// TIA Portal V17 export
// export: Created 2025-03-05T07:59:25.5463254Z, ExportSetting WithDefaults, DisplayName Totally Integrated Automation Portal, DisplayVersion V17 Update 8, DisplayName TIA Portal Openness, DisplayVersion V17 Update 8, DisplayName TIA Portal Version Control Interface, DisplayVersion V17, DisplayName SINAMICS Startdrive Advanced, DisplayVersion V17 SP2, DisplayName SINAMICS Startdrive G110M, G120, G120C, G120D, G120P, G115D, DisplayVersion V17 SP2, DisplayName SINAMICS Startdrive G130, G150, S120, S150, SINAMICS MV, S210, DisplayVersion V17 SP2, DisplayName STEP 7 Professional, DisplayVersion V17 Update 8, DisplayName SINUMERIK ONE STEP 7 Toolbox, DisplayVersion V17 Update 12, DisplayName SINUMERIK 840D sl STEP 7 Toolbox, DisplayVersion V17 Update 12, DisplayName STEP 7 Safety, DisplayVersion V17 Update 6, DisplayName WinCC Advanced, DisplayVersion V17 Update 8
FUNCTION "FC8001_PART_CHANGE" : Void   // FC8001, LAD
{ S7_Optimized_Access := 'FALSE' }
AUTHOR : ETXETAR
VERSION : 1.0
// Change the workpiece code (0x means decimal)
// => input identifier = 0x61 
// 
// When the workpiece code is changed to  317 (317 is entered in input field (5)) 
// on the 3rd station, the following will result:  
// 
// DB59.DBB80:input identifier = 0x61 
// DB59.DBB79: selected station = 0x03 
// DB59.DBW68: Code  = 317 (decimal) 
//  
// 
// Change workpiece status OK/NOK 
// => input ID 0x40, column ID 0x00
// 
// When the status of a workpiece F (= sixth workpiece) is changed at the 3rd 
// station, the following data contents apply:
// DB59.DBB80: Input ID 0x40 + workpiece no. 6 = 0x46
// DB59.DBB79: Selected station 3 = 0x03 
//  
// 
// Change workpiece status exists/does not exist 
// => input ID 0x40, column ID 0x40
// 
// When the status of a workpiece F (= sixth workpiece) is changed at the 3rd 
// station, the following data contents apply:
// DB59.DBB80: Input ID 0x40 + workpiece no. 6 = 0x46
// DB59.DBB79: Column code 0x40 + selected station 3 = 0x43
// stored: AutoNumber false, IsIECCheckEnabled false, SetENOAutomatically false, UDAEnableTagReadback false
   VAR_INPUT
      Plus : Bool;
      Minus : Bool;
      Change_type : Bool;
   END_VAR
   VAR_TEMP
      aux1 : Int;
      DBB79 : Int;
      DBB80 : Int;
      TypBCD : Word;
   END_VAR
BEGIN

NETWORK
TITLE = 
      L     "LTLP_HMIProInterfaceData".noFunctionLow;

      BTI;
      T     #DBB79;
      L     "LTLP_HMIProInterfaceData".noFunctionHigh;
      OPN   "LTLP_HMIProInterfaceData";
      BTI;
      T     #DBB80;

NETWORK
TITLE = Part type change request
      A     #Change_type;
      A(;
      L     #DBB80;
      L     61;
      ==I;
      );
      JCN   ok;
      L     #DBB79;  //Station number
      L     1;  //Station adress (1556,1560,1564)
      -I;
      L     4;
      *I;
      L     1556;
      +I;
      SLW   3;
      LAR1;  //Load pointer Program number
      L     "LTLP_HMIProInterfaceData".codeWorkpiece;  // Load part type decimal
      OPN   "LTLP_HMIProInterfaceData";
      ITB;  //Convert to BCD
      T     #TypBCD;  //Transfer to local
      L     #TypBCD.%B0;  //Load high byte
      T     DBB [AR1, P#0.0];  //Transfer to low byte
      L     #TypBCD.%B1;  //Load low byte
      T     DBB [AR1, P#1.0];  //Transfer to high byte

      L     #DBB79;  //Station number
      L     1;  //Station adress (1556,1560,1564)
      -I;
      L     2;
      *I;
      L     2822;
      +I;
      SLW   3;
      LAR1;
      L     "LTLP_HMIProInterfaceData".codeWorkpiece;
      OPN   "LTLP_HMIProInterfaceData";
      T     DBW [AR1, P#0.0];
      JU    fin1;

REGION Network 3
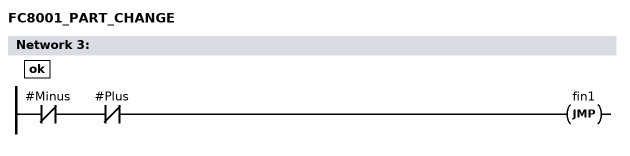
   Label( ok )
   RUNG wire#powerrail
      I_Contact( #Minus )
      I_Contact( #Plus )
      JumpCoil( fin1 )
   END_RUNG
   // the same network as SCL:
   ok:
   IF NOT #Minus AND NOT #Plus THEN GOTO fin1; END_IF;
END_REGION

NETWORK
TITLE = OK/Not OK change request

      L     #DBB79;
      L     40;
      >I;
      JC    pres;
      L     #DBB79;  //Station number
      L     1;  //Station adress (1556,1560,1564)
      -I;
      L     4;
      *I;
      L     1558;  //First OK adress
      +I;
      SLW   3;
      LAR1;  // load pointer

      L     #DBB80;  //part number (up to 8)
      L     40;
      -I;
      T     #aux1;
      L     4;  // if GT 4
      >I;
      JC    may;
      L     #aux1;  //Part number <=4
      L     2;
      *I;
      L     1;
      -I;
      TAR1;
      +I;
      LAR1;
      JU    cam1;
may:  L     1;  //part number >4
      SLW   3;
      +AR1;  //increase pointer 1 byte
      L     #aux1;
      L     2;
      *I;
      L     9;
      -I;
      TAR1;
      +I;
      LAR1;
cam1: A     #Minus;
      R     DBX [AR1, P#0.0];
      A     #Plus;
      S     DBX [AR1, P#0.0];
      JU    fin1;

NETWORK
TITLE = Part present change request

pres: L     #DBB79;
      L     40;
      >I;
      JCN   fin1;
      L     #DBB79;
      L     80;  //Up to 40 stations
      <=I;
      JCN   fin1;
      L     #DBB79;  //Station number
      L     41;  //Station adress (1556,1560,1564)
      -I;
      L     4;
      *I;
      L     1558;  //First OK adress
      +I;
      SLW   3;
      LAR1;  // load pointer

      L     #DBB80;  //part number (up to 8)
      L     40;
      -I;
      T     #aux1;
      L     4;  // if GT 4
      >I;
      JC    may1;
      L     #aux1;  //Part number <=4
      L     2;
      *I;
      L     2;
      -I;
      TAR1;
      +I;
      LAR1;
      JU    cam2;
may1: L     1;  //part number >4
      SLW   3;
      +AR1;  //increase pointer 1 byte
      L     #aux1;
      L     2;
      *I;
      L     10;
      -I;
      TAR1;
      +I;
      LAR1;
cam2: A     #Minus;
      R     DBX [AR1, P#0.0];
      A     #Plus;
      S     DBX [AR1, P#0.0];



NETWORK
TITLE = 
fin1: NOP   0;



END_FUNCTION
